(* CoDeSys 2.3.9.41 project: Aufgabe_2.pro *)
(* Libraries: STANDARD.LIB 5.6.98 11:03:02 *)

(* Task configuration *)
TASK Standard (PRIORITY := 1, INTERVAL := T#5ms);
	Main
END_TASK

(* Global variable list: Global_Variables *)
VAR_GLOBAL
	globalButtonYellow AT%I* : BOOL;
	globalButtonBlue AT%I* : BOOL;
	globalInductiveSensor AT%I* : BOOL;

	intUltrasonicSensor AT%I* : INT;

	globalLightRed AT%Q* : BOOL;
	globalLightGreen AT%Q* : BOOL;

	intAnalogVoltage AT%Q* : INT;

	bufferArray : ARRAY[1.. arrayLength] OF CurrentStatus;

END_VAR

VAR_GLOBAL CONSTANT
	arrayLength : INT := 100;
	F_TASK : INT := 200;
END_VAR

(* Global variable list: TwinCAT_Configuration *)
(* Generated automatically by TwinCAT - (read only) *)
VAR_CONFIG
	.globalButtonYellow AT %IX0.0 : BOOL;	(*  ~ {LinkedWith:TIID^Device 1 (EtherCAT)^Term 1 (EK1200)^Term 2 (EL1004)^Channel 1^Input} *)
	.globalButtonBlue AT %IX0.1 : BOOL;	(*  ~ {LinkedWith:TIID^Device 1 (EtherCAT)^Term 1 (EK1200)^Term 2 (EL1004)^Channel 2^Input} *)
	.globalLightRed AT %QX0.0 : BOOL;	(*  ~ {LinkedWith:TIID^Device 1 (EtherCAT)^Term 1 (EK1200)^Term 3 (EL2004)^Channel 1^Output} *)
	.globalLightGreen AT %QX0.1 : BOOL;	(*  ~ {LinkedWith:TIID^Device 1 (EtherCAT)^Term 1 (EK1200)^Term 3 (EL2004)^Channel 2^Output} *)
END_VAR

(* Data type *)
TYPE CurrentStatus :
STRUCT
	buttonYellow : BOOL;
	buttonBlue : BOOL;
	lightGreen : BOOL;
	lightRed : BOOL;
	inductiveSensor : BOOL;
	intUltrasonicSensor : INT;
	voltageUltrasonicSensor : REAL;
	intAnalogOutput : INT;
	voltageAnalogOutput : REAL;
END_STRUCT
END_TYPE

(* POU MAIN, ST *)
PROGRAM MAIN
VAR
	data0 : SerialDecode;
	data1 : SerialDecode;
	data2 : SerialDecode;
	myarray : ARRAY[0..9] OF REAL;
	i : INT;
	sum : REAL := 0;
	prod : REAL := 1;
	blueEdge : EdgeDetectorDouble;
	yellowEdge : EdgeDetectorDouble;
	myFSM : FSM;
	volt : REAL;
	myfill : fillArray;
	filt_iir : lowpass;
	factor : REAL := 0.9;
	status : CurrentStatus;
	filt_fir : CurrentStatus;
END_VAR
DoSomeMath();

BitShift();

data0(sw := 16#1D06);
data1(sw := 16#534C);
data2(sw := 16#C705);
FOR i := 0 TO 9 BY 1 DO
myarray[i] := i+1;
END_FOR
sum := 0;
prod := 1;
FOR i := 0 TO 9 BY 1 DO
	sum := Addition(sum, myarray[i]);
END_FOR
i := 0;
WHILE i <= 9 DO
	prod := Multiplication(prod, myarray[i]);
	i := i + 1;
END_WHILE

Generator();

blueEdge(inputValue := globalButtonBlue, threshold := 40);
yellowEdge(inputValue := globalButtonYellow, threshold := 40);
globalLightRed:= blueEdge.risingEdge OR yellowEdge.fallingEdge OR yellowEdge.risingEdge OR blueEdge.fallingEdge;
globalLightGreen := yellowEdge.double OR blueEdge.double;

status.buttonBlue := globalButtonBlue;
status.buttonYellow := globalButtonYellow;
status.inductiveSensor := globalInductiveSensor;
status.intUltrasonicSensor := intUltrasonicSensor;
status.voltageUltrasonicSensor := int_to_volt(intUltrasonicSensor);

myFSM();
volt := int_to_volt(intUltrasonicSensor);
myfill(data := status);
filt_iir(data := volt, factor := factor);
filt_fir := ComputeMeanValue();


volt := filt_iir.out;

intAnalogVoltage := volt_to_int(volt);

status.lightGreen := globalLightGreen;
status.lightRed := globalLightRed;
status.voltageAnalogOutput := volt;
status.intAnalogOutput :=intAnalogVoltage;
END_PROGRAM

(* POU SerialDecode, ST *)
FUNCTION_BLOCK SerialDecode
VAR_INPUT
	sw : WORD;
END_VAR
VAR_OUTPUT
	inLength : INT;
	overrunError : BOOL;
	framingError : BOOL;
	parityError : BOOL;
	bufferFull : BOOL;
	initAccepted : BOOL;
	receiveRequest : BOOL;
	transmitAccepted : BOOL;
END_VAR
VAR
END_VAR
inLength := WORD_TO_INT(SHR((sw AND 16#FF00), 8));
overrunError := sw.6;
framingError := sw.5;
parityError := sw.4;
bufferFull := sw.3;
initAccepted := sw.2;
receiveRequest := sw.1;
transmitAccepted := sw.0;
END_FUNCTION_BLOCK

(* POU EdgeDetectorDouble, ST *)
FUNCTION_BLOCK EdgeDetectorDouble
VAR_INPUT
	inputValue : BOOL;
	threshold : INT;
END_VAR
VAR_OUTPUT
	risingEdge : BOOL;
	fallingEdge : BOOL;
	double : BOOL;
END_VAR
VAR
	prev : BOOL := FALSE;
	timer : INT := 0;
END_VAR
IF inputValue > prev THEN
	risingEdge := TRUE;
	fallingEdge := FALSE;
	IF timer < threshold THEN
		double := TRUE;
	ELSE
		double := FALSE;
	END_IF
	timer := 0;
ELSIF inputValue < prev THEN
	risingEdge := FALSE;
	fallingEdge := TRUE;
	IF timer < 32767 THEN
		timer := timer + 1;
	END_IF
	double := FALSE;
ELSE
	risingEdge := FALSE;
	fallingEdge := FALSE;
	IF timer < 32767 THEN
		timer := timer + 1;
	END_IF
	double := FALSE;
END_IF
prev := inputValue;
END_FUNCTION_BLOCK

(* POU FSM, ST *)
FUNCTION_BLOCK FSM
VAR_INPUT
END_VAR
VAR_OUTPUT
END_VAR
VAR
	state : INT := 0;
	bEdge : EdgeDetectorDouble;
	yEdge : EdgeDetectorDouble;
	count : INT := 0;
	led_green : BOOL := FALSE;
	led_red : BOOL := FALSE;
	period : INT := 68;
END_VAR
VAR CONSTANT
	st_off : INT := 0;
	st_blink : INT := 1;
	st_red : INT :=2 ;
	st_green : INT := 3;
END_VAR
bEdge(inputValue := globalButtonBlue, threshold := 40);
yEdge(inputValue := globalButtonYellow, threshold := 40);
CASE state OF
	st_off:
		led_red := FALSE;
		led_green := FALSE;
		IF bEdge.risingEdge = TRUE THEN
			state := st_blink;
			IF bEdge.double = TRUE THEN
				period := 34;
			ELSE
				period := 68;
			END_IF
		ELSIF yEdge.risingEdge = TRUE THEN
			state := st_red;
		END_IF

	st_blink:
		IF count >= period THEN
			count := 0;
			led_red := NOT led_red;
			led_green := NOT led_green;
		ELSE
			count := count + 1;
		END_IF
		IF bEdge.risingEdge = TRUE THEN
			state := st_off;
		ELSIF yEdge.risingEdge = TRUE THEN
			state := st_red;
		END_IF
	st_red:
		led_red := TRUE;
		led_green := FALSE;
		IF bEdge.risingEdge = TRUE THEN
			state := st_blink;
			led_red := FALSE;
			led_green := FALSE;
		ELSIF yEdge.risingEdge = TRUE THEN
			state := st_green;
		END_IF
	st_green:
		led_red := FALSE;
		led_green := TRUE;
		IF bEdge.risingEdge = TRUE THEN
			state := st_blink;
			led_red := FALSE;
			led_green := FALSE;
		ELSIF yEdge.risingEdge = TRUE THEN
			state := st_red;
		END_IF
END_CASE

		globalLightRed :=led_red ;
		globalLightGreen := led_green;
END_FUNCTION_BLOCK

(* POU fillArray, ST *)
FUNCTION_BLOCK fillArray
VAR_INPUT
	data : CurrentStatus;
END_VAR
VAR_OUTPUT
	out: CurrentStatus;
END_VAR
VAR
	i : INT;
END_VAR
IF i < arrayLength THEN
	i := i + 1;
ELSE
	i := 1;
END_IF

out := bufferArray[i] ;
bufferArray[i] := data;
END_FUNCTION_BLOCK

(* POU lowpass, ST *)
FUNCTION_BLOCK lowpass
VAR_INPUT
	data : REAL;
	factor : REAL;
END_VAR
VAR_OUTPUT
	out : REAL;
END_VAR
VAR
	out_buf : REAL := 0;
END_VAR
out_buf := factor * out_buf + (1 - factor) * data;
out := out_buf;
END_FUNCTION_BLOCK

(* POU DoSomeMath, ST *)
PROGRAM DoSomeMath
VAR
	a : REAL := 1;
	b : REAL := 2;
	sum : REAL;
	diff : REAL;
	prod : REAL;
	quot : REAL;
END_VAR
sum := Addition(a:=a, b:=b);
diff := Subtraction(a:=a, b:=b);
prod := Multiplication(a:=a, b:=b);
quot := Division(a:=a, b:=b);
END_PROGRAM

(* POU Addition, ST *)
FUNCTION Addition : REAL
VAR_INPUT
	a : REAL;
	b : REAL;
END_VAR
VAR
END_VAR
Addition := a + b;
END_FUNCTION

(* POU Subtraction, ST *)
FUNCTION Subtraction : REAL
VAR_INPUT
	a : REAL;
	b : REAL;
END_VAR
VAR
END_VAR
Subtraction := a - b;
END_FUNCTION

(* POU Multiplication, ST *)
FUNCTION Multiplication : REAL
VAR_INPUT
	a : REAL;
	b : REAL;
END_VAR
VAR
END_VAR
Multiplication := a * b;
END_FUNCTION

(* POU Division, ST *)
FUNCTION Division : REAL
VAR_INPUT
	a : REAL;
	b : REAL;
END_VAR
VAR
END_VAR
IF b = 0 THEN
	Division := 0;
ELSE
	Division := a / b;
END_IF
END_FUNCTION

(* POU BitShift, ST *)
PROGRAM BitShift
VAR
	myWord : WORD := 16#5D7A;
	shifted_right : WORD;
	shifted_left : DWORD;
	ormask : WORD;
END_VAR
shifted_right := SHR(myword, 3);
shifted_left := SHL(WORD_TO_DWORD(myword),3);
ormask := myword OR 16#F000;
END_PROGRAM

(* POU Generator, ST *)
PROGRAM Generator
VAR
	t : UINT := 0;
	a : REAL := 1;
	offset : REAL := 0;
	w : REAL := 1.0;
	duty : REAL := 0.25;
	sinus : REAL;
	square : REAL;
	pwm : REAL;
END_VAR
IF t <= REAL_TO_INT(w*F_TASK) THEN
	t := t + 1;
ELSE
	t := 0;
END_IF
sinus := SinusFunction(a, offset, w, t);
square := SquareSignal(a, offset, w, t);
pwm := PwmSignal(a, offset, w, t, duty);
END_PROGRAM

(* POU SinusFunction, ST *)
FUNCTION SinusFunction : REAL
VAR_INPUT
	a : REAL;
	offset : REAL;
	w : REAL;
	t : INT;
END_VAR
VAR
END_VAR
SinusFunction := a * SIN(INT_TO_REAL(t)*w /F_TASK *2.0*3.1415) + offset;
END_FUNCTION

(* POU SquareSignal, ST *)
FUNCTION SquareSignal : REAL
VAR_INPUT
	a : REAL;
	offset : REAL;
	w : REAL;
	t : INT;
END_VAR
VAR
	per : INT;
END_VAR
per := REAL_TO_INT(F_TASK / w);
IF (t MOD per) < (per / 2) THEN
	SquareSignal := offset + a;
ELSE
	SquareSignal := offset - a;
END_IF
END_FUNCTION

(* POU PwmSignal, ST *)
FUNCTION PwmSignal : REAL
VAR_INPUT
	a : REAL;
	offset : REAL;
	w : REAL;
	t : INT;
	duty : REAL;
END_VAR
VAR
	per : INT;
END_VAR
per := REAL_TO_INT(F_TASK / w);
IF duty*per >= per THEN
	PwmSignal := offset + a;
ELSIF duty*per <=0 THEN
	PwmSignal := offset - a;
ELSIF (t MOD per) < duty*per THEN
	PwmSignal := offset + a;
ELSE
	PwmSignal := offset - a;
END_IF
END_FUNCTION

(* POU int_to_volt, ST *)
FUNCTION int_to_volt : REAL
VAR_INPUT
	input : INT;
END_VAR
VAR
END_VAR
int_to_volt := 10 - INT_TO_REAL(input) * 10 / 16#7FFF;
END_FUNCTION

(* POU ComputeMeanValue, ST *)
FUNCTION ComputeMeanValue : CurrentStatus
VAR_INPUT
END_VAR
VAR
	i : INT ;
	sum : CurrentStatus;
END_VAR
FOR i := 1 TO arrayLength BY 1 DO
	sum.intAnalogOutput := sum.intAnalogOutput+ bufferArray[i].intAnalogOutput;
	sum.intUltrasonicSensor := sum.intUltrasonicSensor+ bufferArray[i].intUltrasonicSensor;
	sum.voltageAnalogOutput := sum.voltageAnalogOutput+ bufferArray[i].voltageAnalogOutput;
	sum.voltageUltrasonicSensor := sum.voltageUltrasonicSensor+ bufferArray[i].voltageUltrasonicSensor;
END_FOR
ComputeMeanValue.intAnalogOutput := sum.intAnalogOutput / arrayLength;
ComputeMeanValue.intUltrasonicSensor := sum.intUltrasonicSensor / arrayLength;
ComputeMeanValue.voltageAnalogOutput := sum.voltageAnalogOutput / arrayLength;
ComputeMeanValue.voltageUltrasonicSensor := sum.voltageUltrasonicSensor / arrayLength;
END_FUNCTION

(* POU volt_to_int, ST *)
FUNCTION volt_to_int : INT
VAR_INPUT
	input : REAL;
END_VAR
VAR
END_VAR
volt_to_int := REAL_TO_INT(input * 16#7FFF / 10);
END_FUNCTION

(* POU EdgeDetector, ST *)
FUNCTION_BLOCK EdgeDetector
VAR_INPUT
	inputValue : BOOL;
END_VAR
VAR_OUTPUT
	risingEdge : BOOL;
	fallingEdge : BOOL;
END_VAR
VAR
	prev : BOOL := FALSE;
END_VAR
IF inputValue > prev THEN
	risingEdge := TRUE;
	fallingEdge := FALSE;
ELSIF inputValue < prev THEN
	risingEdge := FALSE;
	fallingEdge := TRUE;
ELSE
	risingEdge := FALSE;
	fallingEdge := FALSE;
END_IF
prev := inputValue;
END_FUNCTION_BLOCK
